PROGRAM PRG_TXI_VAC_PUMPS
VAR
	dummy_gauge : ST_VG;
END_VAR

//beamline dummy gauge
dummy_gauge.xPRESS_OK := TRUE;
dummy_gauge.xAT_VAC := TRUE;
dummy_gauge.eState := ValidLo;
dummy_gauge.rPRESS := 1e-4;

//B940-009-R17-PCI-01
fb_TV1K3_PIP_01(i_stGauge := fb_TV1K3_GPI_01.PG, i_xOverrideMode := xSystemOverrideMode1);
fb_ST1K3_PIP_01(i_stGauge := fb_ST1K3_GPI_01.PG, i_xOverrideMode := xSystemOverrideMode1);
fb_PC1K3_PIP_01(i_stGauge := dummy_gauge, i_xOverrideMode := xSystemOverrideMode1);
fb_PC1K3_PIP_02(i_stGauge := dummy_gauge, i_xOverrideMode := xSystemOverrideMode1);

//B940-009-R17-PCI-02
fb_TV2K3_PIP_01(i_stGauge := fb_TV2K3_GPI_01.PG, i_xOverrideMode := xSystemOverrideMode1);
fb_TV3K3_PIP_01(i_stGauge := fb_TV3K3_GPI_01.PG, i_xOverrideMode := xSystemOverrideMode1);
fb_TV4K3_PIP_01(i_stGauge := fb_TV4K3_GPI_01.PG, i_xOverrideMode := xSystemOverrideMode1);

END_PROGRAM

(* stored: Version 1.1.0.1, ProductVersion 3.1.4024.6
   POU PRG_TXI_VAC_PUMPS: Id {582ff63e-8787-478b-bcea-9d2bdf315108}, SpecialFunc None *)
